FUNCTION_BLOCK FB_InterlockControl (* Basic Function Block Type *)
  (* Standard: 61499-2 *)
  (* Version 0.0, 2014-5-4, wildai, nxtControl GmbH, Template *)
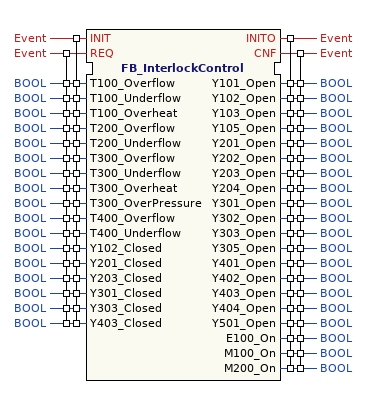
  EVENT_INPUT
    INIT WITH T100_Overflow, T100_Underflow, T100_Overheat, T200_Overflow, T200_Underflow, T300_Overflow, T300_Underflow, T300_Overheat, T300_OverPressure, T400_Overflow, T400_Underflow, Y102_Closed, Y201_Closed, Y203_Closed, Y301_Closed, Y303_Closed, Y403_Closed; (* Initialization Request *)
    REQ WITH T100_Overflow, T100_Underflow, T100_Overheat, T200_Overflow, T200_Underflow, T300_Overflow, T300_Underflow, T300_Overheat, T300_OverPressure, T400_Overflow, T400_Underflow, Y102_Closed, Y201_Closed, Y203_Closed, Y301_Closed, Y303_Closed, Y403_Closed; (* Normal Execution Request *)
  END_EVENT
  EVENT_OUTPUT
    INITO WITH Y101_Open, Y102_Open, Y103_Open, Y105_Open, Y201_Open, Y202_Open, Y203_Open, Y204_Open, Y301_Open, Y302_Open, Y303_Open, Y305_Open, Y401_Open, Y402_Open, Y403_Open, Y404_Open, Y501_Open, E100_On, M100_On, M200_On; (* Initialization Confirm *)
    CNF WITH Y101_Open, Y102_Open, Y103_Open, Y105_Open, Y201_Open, Y202_Open, Y203_Open, Y204_Open, Y301_Open, Y302_Open, Y303_Open, Y305_Open, Y401_Open, Y402_Open, Y403_Open, Y404_Open, Y501_Open, E100_On, M100_On, M200_On; (* Execution Confirmation *)
  END_EVENT
  VAR_INPUT
    T100_Overflow : BOOL;
    T100_Underflow : BOOL;
    T100_Overheat : BOOL;
    T200_Overflow : BOOL;
    T200_Underflow : BOOL;
    T300_Overflow : BOOL;
    T300_Underflow : BOOL;
    T300_Overheat : BOOL;
    T300_OverPressure : BOOL;
    T400_Overflow : BOOL;
    T400_Underflow : BOOL;
    Y102_Closed : BOOL;
    Y201_Closed : BOOL;
    Y203_Closed : BOOL;
    Y301_Closed : BOOL;
    Y303_Closed : BOOL;
    Y403_Closed : BOOL;
  END_VAR
  VAR_OUTPUT
    Y101_Open : BOOL;
    Y102_Open : BOOL;
    Y103_Open : BOOL;
    Y105_Open : BOOL;
    Y201_Open : BOOL;
    Y202_Open : BOOL;
    Y203_Open : BOOL;
    Y204_Open : BOOL;
    Y301_Open : BOOL;
    Y302_Open : BOOL;
    Y303_Open : BOOL;
    Y305_Open : BOOL;
    Y401_Open : BOOL;
    Y402_Open : BOOL;
    Y403_Open : BOOL;
    Y404_Open : BOOL;
    Y501_Open : BOOL;
    E100_On : BOOL;
    M100_On : BOOL;
    M200_On : BOOL;
  END_VAR
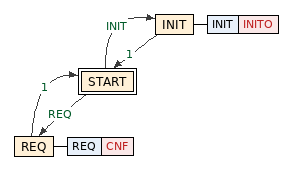
  EC_STATES
    START; (* Initial State *)
    INIT : INIT -> INITO; (* Initialization *)
    REQ : REQ -> CNF; (* Normal execution *)
  END_STATES
  EC_TRANSITIONS
    START TO INIT := INIT;
    INIT TO START := 1;
    START TO REQ := REQ;
    REQ TO START := 1;
  END_TRANSITIONS
  ALGORITHM INIT IN ST: (* Initialization algorithm *)
;

Y101_Open := TRUE;
Y102_Open := TRUE;
Y103_Open := TRUE;
Y105_Open := TRUE;
Y201_Open := TRUE;
Y202_Open := TRUE;
Y203_Open := TRUE;
Y204_Open := TRUE;
Y301_Open := TRUE;
Y302_Open := TRUE;
Y303_Open := TRUE;
Y305_Open := TRUE;
Y401_Open := TRUE;
Y402_Open := TRUE;
Y403_Open := FALSE;
Y404_Open := TRUE;
Y501_Open := TRUE;
E100_On := TRUE;
M100_On := TRUE;
M200_On := TRUE;
  END_ALGORITHM
  ALGORITHM REQ IN ST: (* Normally executed algorithm *)
;

/* Interlocks for Valve, Heater and Pump */
Y101_Open := TRUE;
Y102_Open := TRUE;
Y103_Open := TRUE;
Y105_Open := TRUE;
Y201_Open := TRUE;
Y202_Open := TRUE;
Y203_Open := TRUE;
Y204_Open := TRUE;
Y301_Open := TRUE;
Y302_Open := TRUE;
Y303_Open := TRUE;
Y305_Open := TRUE;
Y401_Open := TRUE;
Y402_Open := TRUE;
Y403_Open := FALSE;
Y404_Open := TRUE;
Y501_Open := TRUE;
E100_On := TRUE;
M100_On := TRUE;
M200_On := TRUE;

IF T100_Overflow OR T400_Underflow THEN
	Y101_Open := FALSE;
END_IF;

IF T100_Underflow THEN
	Y102_Open := FALSE;
END_IF;

IF T100_Underflow OR T300_Overflow THEN
	Y103_Open := FALSE;
END_IF;

IF T100_Underflow THEN
	Y105_Open := FALSE;
END_IF;

IF T200_Underflow THEN
	Y201_Open := FALSE;
END_IF;

IF T200_Underflow THEN
	Y202_Open := FALSE;
END_IF;

IF T200_Overflow THEN
	Y203_Open := FALSE;
END_IF;

IF T200_Overflow OR T300_Underflow THEN
	Y204_Open := FALSE;
END_IF;
IF T300_OverPressure THEN
	Y204_Open := TRUE;
END_IF;

IF T300_Overflow THEN
	Y301_Open := FALSE;
END_IF;

IF T300_Overflow THEN
	Y302_Open := FALSE;
END_IF;

IF T300_Underflow THEN
	Y305_Open := FALSE;
END_IF;

IF T300_Underflow THEN
	Y401_Open := FALSE;
END_IF;

IF T200_Underflow OR T400_Overflow THEN
	Y402_Open := FALSE;
END_IF;

IF T400_Underflow THEN
	Y404_Open := FALSE;
END_IF;

IF T100_Overflow THEN
	Y501_Open := FALSE;
END_IF;

IF T100_Overheat OR T100_Underflow THEN
	E100_On := FALSE;
END_IF;

IF Y102_Closed OR (Y203_Closed AND Y403_Closed) THEN
	M100_On := FALSE;
END_IF;

IF Y301_Closed OR Y303_Closed OR Y201_Closed THEN
	M200_On := FALSE;
END_IF;
  END_ALGORITHM
END_FUNCTION_BLOCK
